VAR_GLOBAL
	FB_UDP_Connection_arr	: ARRAY[0..NR_OF_DRIVEMASTERS] OF FB_UDP_DriveCom;
END_VAR

(* stored: Version 1.1.0.1, ProductVersion 3.1.4024.12
   GVL GVL_FB: Id {1829242d-38ba-4f45-8391-04cfc7edf4d3} *)
